Universal Robots PolyScope program: Group21Lab1Task2.urp

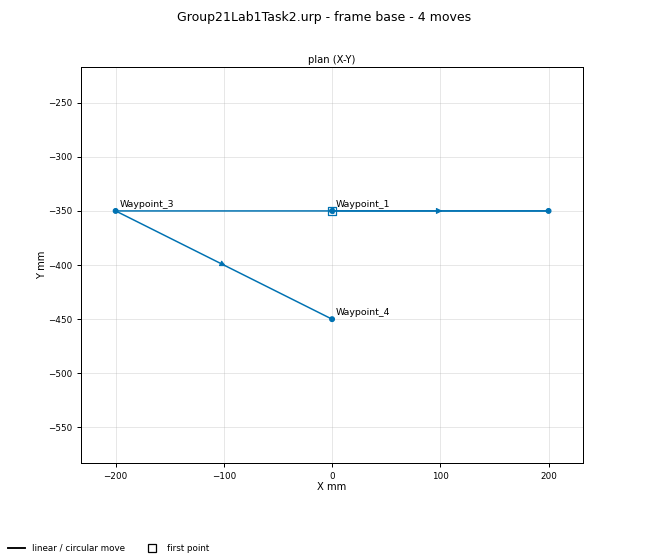
[picture p0: tool path of Group21Lab1Task2.urp in frame base, 4 of 4 moves have a stored position in this frame; points joined in program order, loops and branches not executed]
Program group21p2 (createdIn=3.5.0.10584 lastSavedIn=3.5.0.10584 directory=/programs/usbdisk installation=default robotSerialNumber=2017332505)
Calibrated DH parameters: a=[0, -0.24355, -0.210285, 0.000007, -0.000026, 0]; d=[0.151972, 1.341373, 3.010199, -4.239311, 0.085317, 0.082321]; alpha=[1.570715, -0.004846, 0.008121, 1.57079, -1.571065, 0]; deltaTheta=[0.000017, -0.02667, 0.193133, -0.166555, -0.000046, 0.000042]
Robot Program (runOnlyOnce=false motionType=MoveJ speed=1.047198 acceleration=1.396263 useActiveTCP=false)
  MoveL speed 250 mm/s, acceleration 1200 mm/s^2 (useActiveTCP=false) feature=Base
    Waypoint Waypoint_1: TCP in base x=0.018 y=-350.017 z=199.973 mm, rx=1.6001 ry=0 rz=0.0001 rad; joints [71.731, 19.17, -104.25, -3.287, -90.807, -18.884] deg
    Waypoint Waypoint_2: TCP in base x=199.983 y=-350.001 z=200.028 mm, rx=1.5699 ry=0.0001 rz=0 rad; joints [103.825, 17.078, -88.31, -18.71, -90.129, 13.249] deg
    Waypoint Waypoint_3: TCP in base x=-199.986 y=-350.004 z=200.04 mm, rx=1.5699 ry=0.0002 rz=-0.0001 rad; joints [44.34, 17.126, -88.381, -18.793, -90.149, -46.237] deg
    Waypoint Waypoint_4: TCP in base x=-0.036 y=-449.997 z=200.01 mm, rx=1.5699 ry=0.0002 rz=-0.0002 rad; joints [75.756, 12.108, -70.46, -31.64, -90.077, -14.743] deg
